// TIA Portal V17 export
// export: Created 2025-08-05T09:35:58.6213137Z, ExportSetting WithDefaults, DisplayName Totally Integrated Automation Portal, DisplayVersion V17, DisplayName TIA Portal Openness, DisplayVersion V17, DisplayName TIA Portal Version Control Interface, DisplayVersion V17, DisplayName SINAMICS Startdrive Advanced, DisplayVersion V17, DisplayName SINAMICS Startdrive G130, G150, S120, S150, SINAMICS MV, S210, DisplayVersion V17, DisplayName SINAMICS Startdrive G110M, G120, G120C, G120D, G120P, G115D, DisplayVersion V17, DisplayName STEP 7 Professional, DisplayVersion V17, DisplayName STEP 7 Safety, DisplayVersion V17, DisplayName WinCC Advanced, DisplayVersion V17
DATA_BLOCK "IPG_Weld_Interface_DB"   // DB4
VERSION : 1.0
// stored: AutoNumber true, DBAccessibleFromOPCUA true, DBAccessibleFromWebserver true, InstanceOfName IPG_Weld_Interface, InstanceOfType FB
"IPG_Weld_Interface"
   // VAR_INPUT
   //    iScanner : "Scanner_Inputs";
   //    iYLS : "YLS_Inputs";
   //    iInstance_Index : Int;
   //    iYLR_Power_On : Bool;
   //    bYLR : Bool;
   //    bYLS : Bool;
   // END_VAR
   // VAR_OUTPUT
   //    oScanner : "Scanner_Outputs";
   //    oYLS : "YLS_Outputs";
   //    oYLR_Laser_On : Bool;
   //    oYLR_Reset : Bool;
   // END_VAR
   // VAR
   //    sStep : Int;
   //    sLast_Step : Int;
   //    sScanner_Idle : Bool;
   //    sScanner_Active : Bool;
   //    sScanner_Error : Bool;
   //    sScanner_Waiting_Enable : Bool;
   //    sScanner_Waiting_Strobe : Bool;
   //    sScanner_Waiting_Start : Bool;
   //    tJob_Start_ONS { ExternalAccessible := 'False'; ExternalVisible := 'False'; ExternalWritable := 'False'} : Bool;
   //    tJob_Stop_ONS { ExternalAccessible := 'False'; ExternalVisible := 'False'; ExternalWritable := 'False'} : Bool;
   //    siScanner_Job : Byte;
   //    siScanner_Group : Byte;
   //    soScanner_Job : Byte;
   //    soScanner_Group : Byte;
   //    sVersion { S7_SetPoint := 'True'} : Real;
   //    sStepTimeout : IEC_TIMER;
   //    sReset_Timer { S7_SetPoint := 'True'} : IEC_TIMER;
   //    sLog : Array[0..50] of Struct
   //       Load_Start_Time : Date_And_Time;
   //       Load_Stop_Time : Date_And_Time;
   //       Fire_Start_Time : Date_And_Time;
   //       Fire_Stop_Time : Date_And_Time;
   //       Job_ID : Byte;
   //       Group_ID : Byte;
   //    END_STRUCT;
   //    sBlankLog : Struct
   //       Load_Start_Time : Date_And_Time;
   //       Load_Stop_Time : Date_And_Time;
   //       Fire_Start_Time : Date_And_Time;
   //       Fire_Stop_Time : Date_And_Time;
   //       Job_ID : Byte;
   //       Group_ID : Byte;
   //    END_STRUCT;
   // END_VAR
BEGIN
END_DATA_BLOCK
